FUNCTION_BLOCK EL3204
VAR
	_io : EL3xx4_Data;
	{attribute addProperty Name "WcState"}
	_wcState : WcStateInputToggle;
	{attribute addProperty Name "Info data"}
	_infoData : InfoDataAds;
END_VAR

PROPERTY IO : REFERENCE TO EL3xx4_Data
GET
IO REF= _io;
END_GET
END_PROPERTY

PROPERTY WcState : REFERENCE TO WcStateInputToggle
GET
WcState REF= _wcState;
END_GET
END_PROPERTY

END_FUNCTION_BLOCK

(* stored: Version 1.1.0.1, ProductVersion 3.1.4024.9
   POU EL3204: Id {4a9a89a8-2a3e-01d8-28b1-c044aebffc1d}, SpecialFunc None
   Property IO: Id {c7c4d66e-6fc3-09e1-0690-08bc69089a39}
   Get Get: Id {f1a70f25-fd57-040f-1abb-3e105ca28377}
   Property WcState: Id {8957e421-87ba-0c82-3ed6-2ec22d8805ae}
   Get Get: Id {1279cc3b-51bd-0b87-3426-296c91fd7228} *)
